{attribute 'GeneratedUsingTerminal: EL1918-0000-0016'}
{attribute addProperty BoxType "EL1918-0000-0016"}
{attribute addProperty Id "FSoE_InputsFSoE_Inputs_8E27404E21FSoE_OutputsFSoE_Outputs_5936ECC613"}
{attribute addProperty CRC "2041165480"}
{attribute addProperty Size "34"}
TYPE Module_1_FSOE_79A9B6A8 :
STRUCT
	{attribute addProperty Name "FSoE_Inputs"}
	FSoE_Inputs  : FSoE_Inputs_8E27404E;
	{attribute addProperty Name "FSoE_Outputs"}
	FSoE_Outputs  : FSoE_Outputs_5936ECC6;
END_STRUCT
END_TYPE

(* stored: Version 1.2.0.0, ProductVersion 3.1.4024.9
   DUT Module_1_FSOE_79A9B6A8: Id {f11cf506-496b-4165-bec7-90d0fda52648} *)
